METHOD METH_setMcMoveParams
VAR_INPUT
  stMcMoveParams : ST_mcMoveParams;
  uliMotionIndx  : ULINT;
END_VAR
                  THIS^.stMcMoveParams := stMcMoveParams;
THIS^.uliMotionIndx := uliMotionIndx;

                
END_METHOD

PROPERTY PROP_mcMoveCrcAbs : SM3_Robotics.MC_MoveCircularAbsolute
GET
                    PROP_mcMoveCrcAbs := mcMoveCrcAbs;

                  
END_GET
END_PROPERTY

PROPERTY PROP_mcMoveCrcRel : SM3_Robotics.MC_MoveCircularRelative
GET
                    PROP_mcMoveCrcRel := mcMoveCrcRel;

                  
END_GET
END_PROPERTY

PROPERTY PROP_motionIndx : ULINT
GET
                    PROP_motionIndx := uliMotionIndx;

                  
END_GET
END_PROPERTY

PROPERTY PROP_stMcMoveParams : ST_mcMoveParams
GET
                    PROP_stMcMoveParams := stMcMoveParams;

                  
END_GET
END_PROPERTY

PROPERTY PROP_mcMoveDirAbs : SM3_Robotics.MC_MoveDirectAbsolute
GET
                    PROP_mcMoveDirAbs := mcMoveDirAbs;

                  
END_GET
END_PROPERTY

PROPERTY PROP_mcMoveDirRel : SM3_Robotics.MC_MoveDirectRelative
GET
                    PROP_mcMoveDirRel := mcMoveDirRel;

                  
END_GET
END_PROPERTY

PROPERTY PROP_mcMoveLinAbs : SM3_Robotics.MC_MoveLinearAbsolute
GET
                    PROP_mcMoveLinAbs := mcMoveLinAbs;

                  
END_GET
END_PROPERTY

PROPERTY PROP_mcMoveLinRel : SM3_Robotics.MC_MoveLinearRelative
GET
                    PROP_mcMoveLinRel := mcMoveLinRel;

                  
END_GET
END_PROPERTY
END_FUNCTION_BLOCK

FUNCTION_BLOCK testCFC
VAR
	FB_logAdd_2: FB_logAdd;
END_VAR

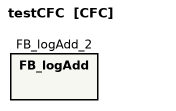
(* CFC diagram, written out as Structured Text *)
FB_logAdd_2();
END_FUNCTION_BLOCK

PROGRAM testFBD
VAR
	FB_logAdd_0: FB_logAdd;
	test : BOOL := TRUE;
END_VAR

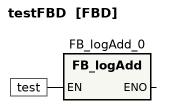
(* FBD diagram, written out as Structured Text *)
FB_logAdd_0(EN := test);
END_PROGRAM

FUNCTION_BLOCK testLD
VAR
  FB_logAdd_1 : FB_logAdd;
  test        : BOOL := TRUE;
END_VAR

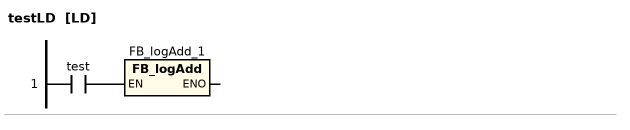
(* LD diagram, written out as Structured Text *)

FB_logAdd_1(EN := test);
END_FUNCTION_BLOCK

FUNCTION_BLOCK testSFC

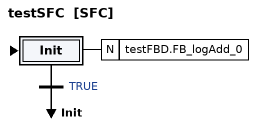
INITIAL_STEP Init:
  testFBD.FB_logAdd_0(N);
END_STEP
TRANSITION FROM Init TO Init
  := TRUE;
END_TRANSITION
END_FUNCTION_BLOCK

PROGRAM POU_DIAG
VAR
END_VAR

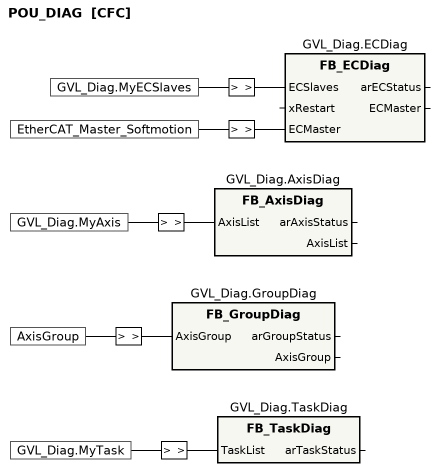
(* CFC diagram, written out as Structured Text *)
GVL_Diag.ECDiag(ECSlaves := GVL_Diag.MyECSlaves, ECMaster := EtherCAT_Master_Softmotion);
GVL_Diag.AxisDiag(AxisList := GVL_Diag.MyAxis);
GVL_Diag.GroupDiag(AxisGroup := AxisGroup);
GVL_Diag.TaskDiag(TaskList := GVL_Diag.MyTask);
END_PROGRAM

PROGRAM Test_ECDiag
VAR
	
	TonTimeout : TON;
	iState : INT;
	// GUI Simulation Flags
	xGuiRestartEC : BOOL;
	sECError : STRING;
	
END_VAR

            
//----------------------------
// Call FUB EtherCat Diagnosis
//----------------------------
(*ECDiag(
		ECMaster := EtherCat_Master_Softmotion,  // Local EtherCAT Master instance
		ECSlaves := MyECSlaves					// Input from MyECSlaves
	  );

*)
//--------------------------------
// Check the status of EtherCAT 
//--------------------------------
CASE iState OF
	 
	// EC Master should be ready in 10 sec
	0: 	TonTimeOut(IN := TRUE,PT := T#10S);   
		IF TonTimeOut.Q THEN
			TonTimeOut(IN := FALSE);
			iState := 1000;  // -> Error evaluation
 		END_IF
	 
		// EC Status ok ?
		IF ECDiag.arECStatus.xEC_OK THEN
			TonTimeOut(IN := FALSE);
			iState := 10;
		END_IF
	
		 
	// EtherCAt is running. Check if an error occurs. 
	10:	IF NOT ECDiag.arECStatus.xEC_OK THEN
			iState := 1000; // -> Error evaluation
		END_IF	

	// Wait for a possible restart EC Master . In this case restart from GUI with variable xGuiRestart	 
	20:	 IF xGuiRestartEC  THEN
			xGuiRestartEC := FALSE;			
			EtherCat_Master_Softmotion.xRestart := TRUE;
			iState := 30;
		END_IF
		
	// Reset Restart Flag		
	30: EtherCat_Master_Softmotion.xRestart := FALSE;
		iState := 0;
	
			
	//  EC Error evaluation
	1000:  
		CASE ECDiag.arECStatus.ErrorID OF
			// Check Slaves. Possibly missing voltage of the regulator. Then restart with xGUIRestartEC
			ECDiagError.Missing_Slaves : iState := 20;
			// Check Slaves. Possibly missing voltage of the regulator. Then restart with xGUIRestartEC
			ECDiagError.Error_in_Slave : iState := 20; 
			// Critical Error in EtherCAT Stack. Check Hardware. 
			ECDiagError.EC_Master_Error: iState := 1000;  
			// replace wrong slave.  
			ECDiagError.Wrong_Slave_Detected : iState := 1000;
  		  ELSE
			// Unknown Error. only possible with a wrong enum list
		 END_CASE

END_CASE


          
END_PROGRAM

PROGRAM PLC_PRG
VAR CONSTANT
  uiNumOfWaypts : UINT := 4;
END_VAR
VAR
  fbMachine : FB_machine(rAxisGrpRefSm3:=AppAxisGroup,
                         sGrpName:='AppAxisGroup',
                         sAxisNames:='A1,A2,A3,A4,A5,A6'); // comma delimted string

  diIndx          : DINT := 0;
  smcPosRef       : SM3_Robotics.SMC_POS_REF;
  stMoveDirParams : ST_moveDirParams;
  stMcMoveParams  : ST_mcMoveParams;

	fbMcMoveElem1 : FB_mcMoveElement;
	fbMcMoveElem2 : FB_mcMoveElement;
	fbMcMoveElem3 : FB_mcMoveElement;
	
	itfMcMoveElem : I_mcMoveElement;
  mcMoveLinkedList : COL.LinkedList;

  stHaltParams : ST_haltParams;

  xMotionFinished : BOOL;
  xHaltFinished   : BOOL;
	
	test : UDINT;
END_VAR

                    // POU_Depictor();
// POU_BoxProperties();
// POU_BasicMotion();

IF diIndx = 0 THEN
  FOR diIndx := 1 TO 3 BY 1 DO
    smcPosRef.a.a0 := DINT_TO_LREAL(diIndx + 1);
    smcPosRef.a.a1 := DINT_TO_LREAL(diIndx + 1);
    smcPosRef.a.a2 := DINT_TO_LREAL(diIndx + 1);
    smcPosRef.a.a3 := DINT_TO_LREAL(diIndx + 1);
    smcPosRef.a.a4 := DINT_TO_LREAL(diIndx + 1);
    smcPosRef.a.a5 := DINT_TO_LREAL(diIndx + 1);

    stMoveDirParams.smcPosRef := smcPosRef;
    stMoveDirParams.smcPtpTyp := SM3_Robotics.SMC_PTP_MOVEMENT_TYPE.Fast;
    stMoveDirParams.smcCrdSys := SM3_Robotics.SMC_COORD_SYSTEM.ACS;

    stMcMoveParams.eMcMotionFbType := E_mcMotionFbType.moveDirAbs;
    stMcMoveParams.stMoveDirParams := stMoveDirParams;

    IF diIndx = 1 THEN
      fbMcMoveElem1(stMcMoveParams:=stMcMoveParams,
                    uliMotionIndx:=DINT_TO_ULINT(diIndx + 1));

      itfMcMoveElem := fbMcMoveElem1;
    ELSIF diIndx = 2 THEN
      fbMcMoveElem2(stMcMoveParams:=stMcMoveParams,
                    uliMotionIndx:=DINT_TO_ULINT(diIndx + 1));

      itfMcMoveElem := fbMcMoveElem2;
    ELSIF diIndx = 3 THEN
      fbMcMoveElem3(stMcMoveParams:=stMcMoveParams,
                    uliMotionIndx:=DINT_TO_ULINT(diIndx + 1));

      itfMcMoveElem := fbMcMoveElem3;
    END_IF

    mcMoveLinkedList.AddElement(itfMcMoveElem);

    test := mcMoveLinkedList.CountElements();
  END_FOR
END_IF

fbMachine.METH_grpPwrOn();
fbMachine.METH_groupEnable();
fbMachine.METH_moveToPosition(mcMoveLinkedList:=mcMoveLinkedList,
                              xMotionFinished=>xMotionFinished);

// IF diIndx2 = 1 THEN
//   fbMachine.METH_groupHalt(stHaltParams:=stHaltParams,
//                            xHaltFinished=>xHaltFinished);
// 
//   IF xHaltFinished THEN
//     diIndx2 := diIndx2 + 1;
//   END_IF
// ELSE
//   IF xMotionFinished AND (diIndx2 < UPPER_BOUND(arrstMcMoveParams, 1)) THEN
//     diIndx2 := diIndx2 + 1;
//   END_IF
// END_IF

// IF diIndx2 >= UPPER_BOUND(arrstMcMoveParams, 1) THEN
//   fbMachine.METH_groupDisable();
//   fbMachine.METH_grpPwrOn();
// END_IF

                  
END_PROGRAM

PROGRAM POU_Depictor
VAR
  depictorCW40 : CW40.Coboworx_Depictor_Data;

  depFrameTCP       : DepictorBase.DepictorFrame;
  ActiveCoordSystem : SMC_COORD_SYSTEM := SMC_COORD_SYSTEM.MCS;
END_VAR

                    depictorCW40(AxisGroup:=AppAxisGroup, axes=>);

                  
END_PROGRAM

PROGRAM POU_BasicMotion
VAR
  mcGrpReadActualPos : SM3_Robotics.MC_GroupReadActualPosition;

  mcGrpEnable : SM3_Robotics.MC_GroupEnable;
  smcGrpPower : SM3_Robotics.SMC_GroupPower;

  smcPosRef    : SM3_Robotics.SMC_POS_REF;
  smcCrdSys    : SM3_Robotics.SMC_COORD_SYSTEM;
  mcMoveLinAbs : SM3_Robotics.MC_MoveLinearAbsolute;
  smcPtpType   : SM3_Robotics.SMC_PTP_MOVEMENT_TYPE;
  mcMoveDirAbs : SM3_Robotics.MC_MoveDirectAbsolute;

  xError     : BOOL;
  smcErrorId : SM3_Error.SMC_ERROR;

  // 	test : SM3_Robotics.AXIS_GROUP_REF_SM3;
  // 	test2 : SM3_Basic.IAxisRef;
  // 	test3 : UDINT;
END_VAR

                    mcGrpReadActualPos(AxisGroup:=AppAxisGroup,
                   Enable:=TRUE,
                   CoordSystem:=SMC_COORD_SYSTEM.MCS);

// test := AppAxisGroup;
// test2 := test.m_aAxes[0];
// test3 := test.m_nNumAxes;

IF NOT A1.bRegulatorRealState THEN
  smcGrpPower(AxisGroup:=AppAxisGroup,
              Enable:=TRUE,
              bRegulatorOn:=TRUE,
              bDriveStart:=TRUE,
              Error=>xError,
              ErrorID=>smcErrorId);
END_IF

// AppAxisGroup.m_state; SM3_Robotics.SMC_AXIS_GROUP_STATE

IF A1.bRegulatorRealState AND
   NOT mcGrpEnable.Done THEN
  mcGrpEnable(AxisGroup:=AppAxisGroup,
              Execute:=TRUE,
              Error=>xError,
              ErrorID=>smcErrorId);
END_IF

IF mcGrpEnable.Done AND
   A1.bRegulatorRealState THEN

  IF NOT mcMoveDirAbs.Done THEN
    smcCrdSys := SM3_Robotics.SMC_COORD_SYSTEM.ACS;

    smcPosRef.a.a0 := 1;
    smcPosRef.a.a1 := 1;
    smcPosRef.a.a2 := 1;
    smcPosRef.a.a3 := 1;
    smcPosRef.a.a4 := 1;
    smcPosRef.a.a5 := 1;

    mcMoveDirAbs(AxisGroup:=AppAxisGroup,
                 Execute:=TRUE,
                 Position:=smcPosRef,
                 MovementType:=smcPtpType,
                 CoordSystem:=smcCrdSys,
                 Error=>xError,
                 ErrorID=>smcErrorId);

    //   IF mcMoveDirAbs.Done THEN
    //     mcMoveDirAbs(AxisGroup:=AppAxisGroup,
    //                  Execute:=FALSE);
    //   END_IF
  ELSIF NOT xError THEN
    smcCrdSys := SM3_Robotics.SMC_COORD_SYSTEM.MCS;

    smcPosRef.c.X := POU_BoxProperties.PosX;
    smcPosRef.c.Y := POU_BoxProperties.PosY;
    smcPosRef.c.Z := POU_BoxProperties.PosZ;
    smcPosRef.c.A := 0;
    smcPosRef.c.B := 90;
    smcPosRef.c.C := 0;

    mcMoveLinAbs(AxisGroup:=AppAxisGroup,
                 Execute:=TRUE,
                 Position:=smcPosRef,
                 Velocity:=A1.fSWMaxVelocity,
                 Acceleration:=A1.fSWMaxAcceleration,
                 Deceleration:=A1.fSWMaxDeceleration,
                 Jerk:=A1.fSWMaxJerk,
                 CoordSystem:=smcCrdSys,
                 Error=>xError,
                 ErrorID=>smcErrorId);

    //   IF mcMoveLinAbs.Done THEN
    //     mcMoveLinAbs(AxisGroup:=AppAxisGroup,
    //                  Execute:=FALSE);
    //   END_IF
  END_IF

END_IF

                  
END_PROGRAM

PROGRAM POU_BoxProperties
VAR
  Length, Height, Width : LREAL := 10;
  //The position is the box' center relative to the World Coordinate System, which is at the base of the robot!
  PosX : LREAL := 750;
  PosY : LREAL := 0;
  PosZ : LREAL := 750;
END_VAR

                    
                  
END_PROGRAM

CONFIGURATION Device
  RESOURCE Application ON PLC
    TASK MainTask(INTERVAL := T#4ms, PRIORITY := 1);
    TASK SoftMotion_PlanningTask(INTERVAL := T#2ms, PRIORITY := 15);
    PROGRAM PLC_PRG WITH MainTask : PLC_PRG;
  END_RESOURCE
END_CONFIGURATION

CONFIGURATION SoftMotion General Axis Pool
END_CONFIGURATION

CONFIGURATION A1
END_CONFIGURATION

CONFIGURATION A2
END_CONFIGURATION

CONFIGURATION A3
END_CONFIGURATION

CONFIGURATION A4
END_CONFIGURATION

CONFIGURATION A5
END_CONFIGURATION

CONFIGURATION A6
END_CONFIGURATION
